// TIA Portal V17 export
// export: Created 2025-03-05T08:01:46.0565803Z, ExportSetting WithDefaults, DisplayName Totally Integrated Automation Portal, DisplayVersion V17 Update 8, DisplayName TIA Portal Openness, DisplayVersion V17 Update 8, DisplayName TIA Portal Version Control Interface, DisplayVersion V17, DisplayName SINAMICS Startdrive Advanced, DisplayVersion V17 SP2, DisplayName SINAMICS Startdrive G110M, G120, G120C, G120D, G120P, G115D, DisplayVersion V17 SP2, DisplayName SINAMICS Startdrive G130, G150, S120, S150, SINAMICS MV, S210, DisplayVersion V17 SP2, DisplayName STEP 7 Professional, DisplayVersion V17 Update 8, DisplayName SINUMERIK ONE STEP 7 Toolbox, DisplayVersion V17 Update 12, DisplayName SINUMERIK 840D sl STEP 7 Toolbox, DisplayVersion V17 Update 12, DisplayName STEP 7 Safety, DisplayVersion V17 Update 6, DisplayName WinCC Advanced, DisplayVersion V17 Update 8
FUNCTION "FC7240_MACHINE_DEVICE_ENABLE_DISABLE" : Void   // FC7240, LAD
{ S7_Optimized_Access := 'FALSE' }
AUTHOR : ETXETAR
VERSION : 1.0
// stored: AutoNumber false, IsIECCheckEnabled false, SetENOAutomatically false, UDAEnableTagReadback false
BEGIN

REGION Network 1: OPTIONS OFF
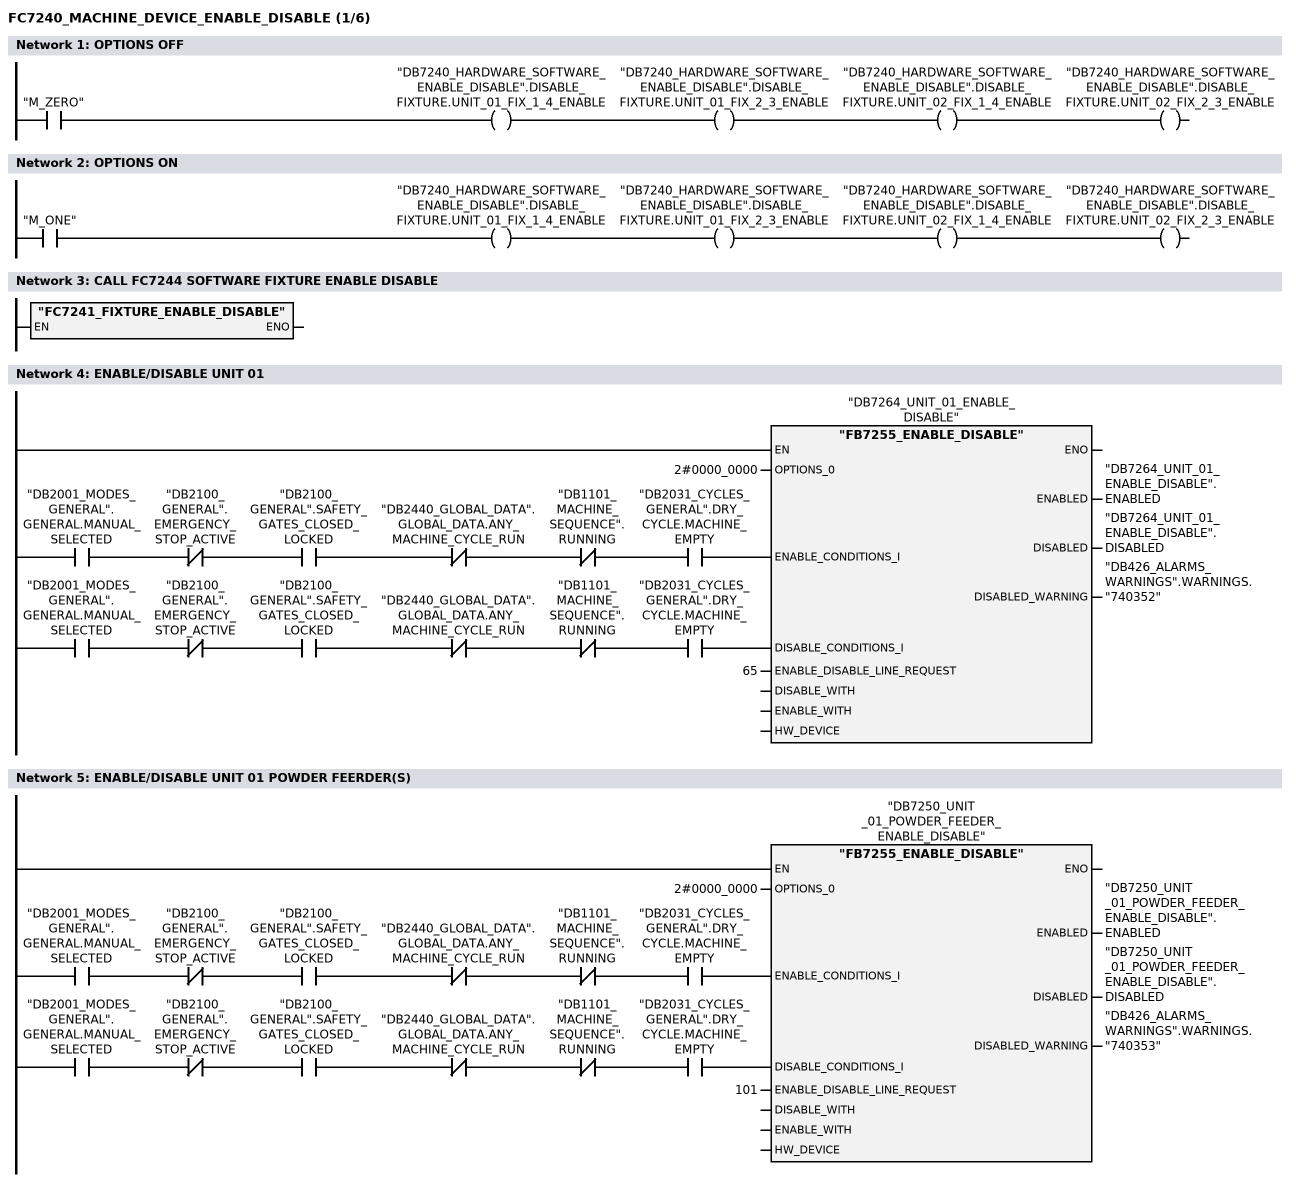
   RUNG wire#powerrail
      Contact( "M_ZERO" )
      Coil( "DB7240_HARDWARE_SOFTWARE_ENABLE_DISABLE".DISABLE_FIXTURE.UNIT_01_FIX_1_4_ENABLE )
      Coil( "DB7240_HARDWARE_SOFTWARE_ENABLE_DISABLE".DISABLE_FIXTURE.UNIT_01_FIX_2_3_ENABLE )
      Coil( "DB7240_HARDWARE_SOFTWARE_ENABLE_DISABLE".DISABLE_FIXTURE.UNIT_02_FIX_1_4_ENABLE )
      Coil( "DB7240_HARDWARE_SOFTWARE_ENABLE_DISABLE".DISABLE_FIXTURE.UNIT_02_FIX_2_3_ENABLE )
   END_RUNG
   // the same network as SCL:
   "DB7240_HARDWARE_SOFTWARE_ENABLE_DISABLE".DISABLE_FIXTURE.UNIT_01_FIX_1_4_ENABLE := "M_ZERO";
   "DB7240_HARDWARE_SOFTWARE_ENABLE_DISABLE".DISABLE_FIXTURE.UNIT_01_FIX_2_3_ENABLE := "M_ZERO";
   "DB7240_HARDWARE_SOFTWARE_ENABLE_DISABLE".DISABLE_FIXTURE.UNIT_02_FIX_1_4_ENABLE := "M_ZERO";
   "DB7240_HARDWARE_SOFTWARE_ENABLE_DISABLE".DISABLE_FIXTURE.UNIT_02_FIX_2_3_ENABLE := "M_ZERO";
END_REGION

REGION Network 2: OPTIONS ON
   RUNG wire#powerrail
      Contact( "M_ONE" )
      Coil( "DB7240_HARDWARE_SOFTWARE_ENABLE_DISABLE".DISABLE_FIXTURE.UNIT_01_FIX_1_4_ENABLE )
      Coil( "DB7240_HARDWARE_SOFTWARE_ENABLE_DISABLE".DISABLE_FIXTURE.UNIT_01_FIX_2_3_ENABLE )
      Coil( "DB7240_HARDWARE_SOFTWARE_ENABLE_DISABLE".DISABLE_FIXTURE.UNIT_02_FIX_1_4_ENABLE )
      Coil( "DB7240_HARDWARE_SOFTWARE_ENABLE_DISABLE".DISABLE_FIXTURE.UNIT_02_FIX_2_3_ENABLE )
   END_RUNG
   // the same network as SCL:
   "DB7240_HARDWARE_SOFTWARE_ENABLE_DISABLE".DISABLE_FIXTURE.UNIT_01_FIX_1_4_ENABLE := "M_ONE";
   "DB7240_HARDWARE_SOFTWARE_ENABLE_DISABLE".DISABLE_FIXTURE.UNIT_01_FIX_2_3_ENABLE := "M_ONE";
   "DB7240_HARDWARE_SOFTWARE_ENABLE_DISABLE".DISABLE_FIXTURE.UNIT_02_FIX_1_4_ENABLE := "M_ONE";
   "DB7240_HARDWARE_SOFTWARE_ENABLE_DISABLE".DISABLE_FIXTURE.UNIT_02_FIX_2_3_ENABLE := "M_ONE";
END_REGION

REGION Network 3: CALL FC7244 SOFTWARE FIXTURE ENABLE DISABLE
   RUNG wire#powerrail
      "FC7241_FIXTURE_ENABLE_DISABLE"()
   END_RUNG
   // the same network as SCL:
   "FC7241_FIXTURE_ENABLE_DISABLE"();
END_REGION

REGION Network 4: ENABLE/DISABLE UNIT 01
   RUNG wire#powerrail
      "DB7264_UNIT_01_ENABLE_DISABLE"(ENABLE_CONDITIONS_I := wire#w1, DISABLE_CONDITIONS_I := wire#w2, OPTIONS_0 := 2#0000_0000, ENABLE_DISABLE_LINE_REQUEST := 65, DISABLE_WITH :=, ENABLE_WITH :=, HW_DEVICE :=, ENABLED => "DB7264_UNIT_01_ENABLE_DISABLE".ENABLED, DISABLED => "DB7264_UNIT_01_ENABLE_DISABLE".DISABLED, DISABLED_WARNING => "DB426_ALARMS_WARNINGS".WARNINGS."740352")
   END_RUNG
   RUNG wire#powerrail
      Contact( "DB2001_MODES_GENERAL".GENERAL.MANUAL_SELECTED )
      I_Contact( "DB2100_GENERAL".EMERGENCY_STOP_ACTIVE )
      Contact( "DB2100_GENERAL".SAFETY_GATES_CLOSED_LOCKED )
      I_Contact( "DB2440_GLOBAL_DATA".GLOBAL_DATA.ANY_MACHINE_CYCLE_RUN )
      I_Contact( "DB1101_MACHINE_SEQUENCE".RUNNING )
      Contact( "DB2031_CYCLES_GENERAL".DRY_CYCLE.MACHINE_EMPTY )
   END_RUNG wire#w1
   RUNG wire#powerrail
      Contact( "DB2001_MODES_GENERAL".GENERAL.MANUAL_SELECTED )
      I_Contact( "DB2100_GENERAL".EMERGENCY_STOP_ACTIVE )
      Contact( "DB2100_GENERAL".SAFETY_GATES_CLOSED_LOCKED )
      I_Contact( "DB2440_GLOBAL_DATA".GLOBAL_DATA.ANY_MACHINE_CYCLE_RUN )
      I_Contact( "DB1101_MACHINE_SEQUENCE".RUNNING )
      Contact( "DB2031_CYCLES_GENERAL".DRY_CYCLE.MACHINE_EMPTY )
   END_RUNG wire#w2
   // the same network as SCL:
   "DB7264_UNIT_01_ENABLE_DISABLE"(OPTIONS_0 := 2#0000_0000,   // "FB7255_ENABLE_DISABLE"
                           ENABLE_CONDITIONS_I := "DB2001_MODES_GENERAL".GENERAL.MANUAL_SELECTED AND NOT "DB2100_GENERAL".EMERGENCY_STOP_ACTIVE AND "DB2100_GENERAL".SAFETY_GATES_CLOSED_LOCKED AND NOT "DB2440_GLOBAL_DATA".GLOBAL_DATA.ANY_MACHINE_CYCLE_RUN AND NOT "DB1101_MACHINE_SEQUENCE".RUNNING AND "DB2031_CYCLES_GENERAL".DRY_CYCLE.MACHINE_EMPTY,
                           DISABLE_CONDITIONS_I := "DB2001_MODES_GENERAL".GENERAL.MANUAL_SELECTED AND NOT "DB2100_GENERAL".EMERGENCY_STOP_ACTIVE AND "DB2100_GENERAL".SAFETY_GATES_CLOSED_LOCKED AND NOT "DB2440_GLOBAL_DATA".GLOBAL_DATA.ANY_MACHINE_CYCLE_RUN AND NOT "DB1101_MACHINE_SEQUENCE".RUNNING AND "DB2031_CYCLES_GENERAL".DRY_CYCLE.MACHINE_EMPTY,
                           ENABLE_DISABLE_LINE_REQUEST := 65,
                           ENABLED => "DB7264_UNIT_01_ENABLE_DISABLE".ENABLED,
                           DISABLED => "DB7264_UNIT_01_ENABLE_DISABLE".DISABLED,
                           DISABLED_WARNING => "DB426_ALARMS_WARNINGS".WARNINGS."740352");
END_REGION

REGION Network 5: ENABLE/DISABLE UNIT 01 POWDER FEERDER(S)
   RUNG wire#powerrail
      "DB7250_UNIT _01_POWDER_FEEDER_ENABLE_DISABLE"(ENABLE_CONDITIONS_I := wire#w1, DISABLE_CONDITIONS_I := wire#w2, OPTIONS_0 := 2#0000_0000, ENABLE_DISABLE_LINE_REQUEST := 101, DISABLE_WITH :=, ENABLE_WITH :=, HW_DEVICE :=, ENABLED => "DB7250_UNIT _01_POWDER_FEEDER_ENABLE_DISABLE".ENABLED, DISABLED => "DB7250_UNIT _01_POWDER_FEEDER_ENABLE_DISABLE".DISABLED, DISABLED_WARNING => "DB426_ALARMS_WARNINGS".WARNINGS."740353")
   END_RUNG
   RUNG wire#powerrail
      Contact( "DB2001_MODES_GENERAL".GENERAL.MANUAL_SELECTED )
      I_Contact( "DB2100_GENERAL".EMERGENCY_STOP_ACTIVE )
      Contact( "DB2100_GENERAL".SAFETY_GATES_CLOSED_LOCKED )
      I_Contact( "DB2440_GLOBAL_DATA".GLOBAL_DATA.ANY_MACHINE_CYCLE_RUN )
      I_Contact( "DB1101_MACHINE_SEQUENCE".RUNNING )
      Contact( "DB2031_CYCLES_GENERAL".DRY_CYCLE.MACHINE_EMPTY )
   END_RUNG wire#w1
   RUNG wire#powerrail
      Contact( "DB2001_MODES_GENERAL".GENERAL.MANUAL_SELECTED )
      I_Contact( "DB2100_GENERAL".EMERGENCY_STOP_ACTIVE )
      Contact( "DB2100_GENERAL".SAFETY_GATES_CLOSED_LOCKED )
      I_Contact( "DB2440_GLOBAL_DATA".GLOBAL_DATA.ANY_MACHINE_CYCLE_RUN )
      I_Contact( "DB1101_MACHINE_SEQUENCE".RUNNING )
      Contact( "DB2031_CYCLES_GENERAL".DRY_CYCLE.MACHINE_EMPTY )
   END_RUNG wire#w2
   // the same network as SCL:
   "DB7250_UNIT _01_POWDER_FEEDER_ENABLE_DISABLE"(OPTIONS_0 := 2#0000_0000,   // "FB7255_ENABLE_DISABLE"
                           ENABLE_CONDITIONS_I := "DB2001_MODES_GENERAL".GENERAL.MANUAL_SELECTED AND NOT "DB2100_GENERAL".EMERGENCY_STOP_ACTIVE AND "DB2100_GENERAL".SAFETY_GATES_CLOSED_LOCKED AND NOT "DB2440_GLOBAL_DATA".GLOBAL_DATA.ANY_MACHINE_CYCLE_RUN AND NOT "DB1101_MACHINE_SEQUENCE".RUNNING AND "DB2031_CYCLES_GENERAL".DRY_CYCLE.MACHINE_EMPTY,
                           DISABLE_CONDITIONS_I := "DB2001_MODES_GENERAL".GENERAL.MANUAL_SELECTED AND NOT "DB2100_GENERAL".EMERGENCY_STOP_ACTIVE AND "DB2100_GENERAL".SAFETY_GATES_CLOSED_LOCKED AND NOT "DB2440_GLOBAL_DATA".GLOBAL_DATA.ANY_MACHINE_CYCLE_RUN AND NOT "DB1101_MACHINE_SEQUENCE".RUNNING AND "DB2031_CYCLES_GENERAL".DRY_CYCLE.MACHINE_EMPTY,
                           ENABLE_DISABLE_LINE_REQUEST := 101,
                           ENABLED => "DB7250_UNIT _01_POWDER_FEEDER_ENABLE_DISABLE".ENABLED,
                           DISABLED => "DB7250_UNIT _01_POWDER_FEEDER_ENABLE_DISABLE".DISABLED,
                           DISABLED_WARNING => "DB426_ALARMS_WARNINGS".WARNINGS."740353");
END_REGION

REGION Network 6: ENABLE/DISABLE UNIT 01 PYROMETER
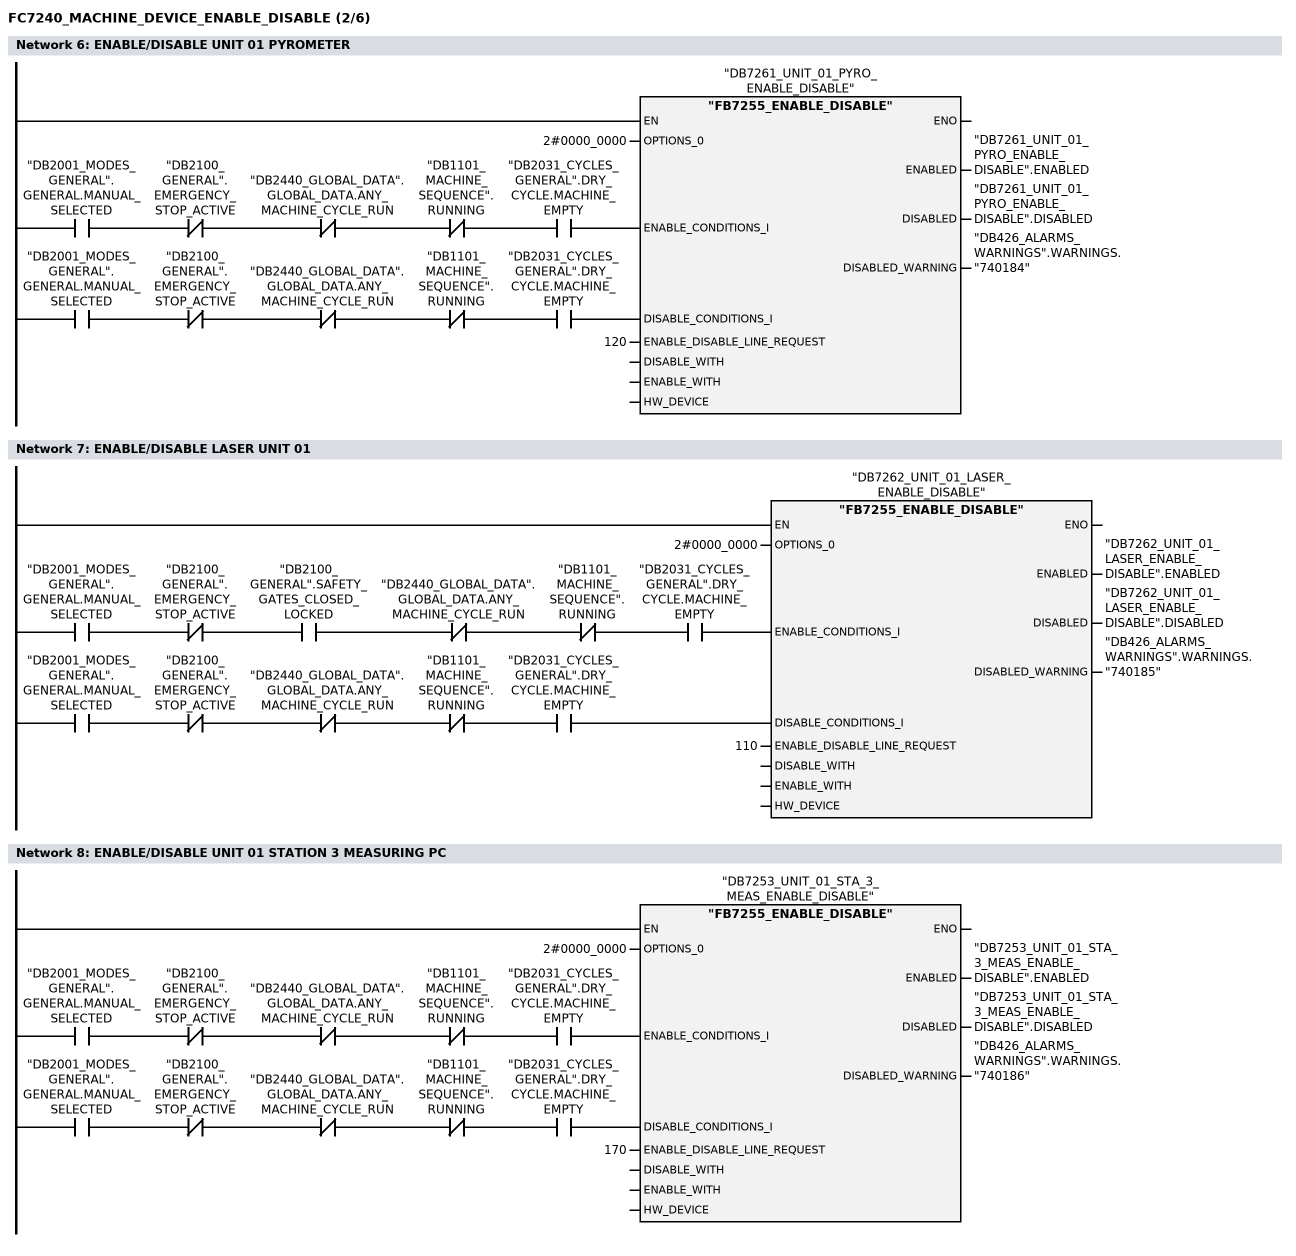
   RUNG wire#powerrail
      "DB7261_UNIT_01_PYRO_ENABLE_DISABLE"(ENABLE_CONDITIONS_I := wire#w1, DISABLE_CONDITIONS_I := wire#w2, OPTIONS_0 := 2#0000_0000, ENABLE_DISABLE_LINE_REQUEST := 120, DISABLE_WITH :=, ENABLE_WITH :=, HW_DEVICE :=, ENABLED => "DB7261_UNIT_01_PYRO_ENABLE_DISABLE".ENABLED, DISABLED => "DB7261_UNIT_01_PYRO_ENABLE_DISABLE".DISABLED, DISABLED_WARNING => "DB426_ALARMS_WARNINGS".WARNINGS."740184")
   END_RUNG
   RUNG wire#powerrail
      Contact( "DB2001_MODES_GENERAL".GENERAL.MANUAL_SELECTED )
      I_Contact( "DB2100_GENERAL".EMERGENCY_STOP_ACTIVE )
      I_Contact( "DB2440_GLOBAL_DATA".GLOBAL_DATA.ANY_MACHINE_CYCLE_RUN )
      I_Contact( "DB1101_MACHINE_SEQUENCE".RUNNING )
      Contact( "DB2031_CYCLES_GENERAL".DRY_CYCLE.MACHINE_EMPTY )
   END_RUNG wire#w1
   RUNG wire#powerrail
      Contact( "DB2001_MODES_GENERAL".GENERAL.MANUAL_SELECTED )
      I_Contact( "DB2100_GENERAL".EMERGENCY_STOP_ACTIVE )
      I_Contact( "DB2440_GLOBAL_DATA".GLOBAL_DATA.ANY_MACHINE_CYCLE_RUN )
      I_Contact( "DB1101_MACHINE_SEQUENCE".RUNNING )
      Contact( "DB2031_CYCLES_GENERAL".DRY_CYCLE.MACHINE_EMPTY )
   END_RUNG wire#w2
   // the same network as SCL:
   "DB7261_UNIT_01_PYRO_ENABLE_DISABLE"(OPTIONS_0 := 2#0000_0000,   // "FB7255_ENABLE_DISABLE"
                           ENABLE_CONDITIONS_I := "DB2001_MODES_GENERAL".GENERAL.MANUAL_SELECTED AND NOT "DB2100_GENERAL".EMERGENCY_STOP_ACTIVE AND NOT "DB2440_GLOBAL_DATA".GLOBAL_DATA.ANY_MACHINE_CYCLE_RUN AND NOT "DB1101_MACHINE_SEQUENCE".RUNNING AND "DB2031_CYCLES_GENERAL".DRY_CYCLE.MACHINE_EMPTY,
                           DISABLE_CONDITIONS_I := "DB2001_MODES_GENERAL".GENERAL.MANUAL_SELECTED AND NOT "DB2100_GENERAL".EMERGENCY_STOP_ACTIVE AND NOT "DB2440_GLOBAL_DATA".GLOBAL_DATA.ANY_MACHINE_CYCLE_RUN AND NOT "DB1101_MACHINE_SEQUENCE".RUNNING AND "DB2031_CYCLES_GENERAL".DRY_CYCLE.MACHINE_EMPTY,
                           ENABLE_DISABLE_LINE_REQUEST := 120,
                           ENABLED => "DB7261_UNIT_01_PYRO_ENABLE_DISABLE".ENABLED,
                           DISABLED => "DB7261_UNIT_01_PYRO_ENABLE_DISABLE".DISABLED,
                           DISABLED_WARNING => "DB426_ALARMS_WARNINGS".WARNINGS."740184");
END_REGION

REGION Network 7: ENABLE/DISABLE LASER UNIT 01
   RUNG wire#powerrail
      "DB7262_UNIT_01_LASER_ENABLE_DISABLE"(ENABLE_CONDITIONS_I := wire#w1, DISABLE_CONDITIONS_I := wire#w2, OPTIONS_0 := 2#0000_0000, ENABLE_DISABLE_LINE_REQUEST := 110, DISABLE_WITH :=, ENABLE_WITH :=, HW_DEVICE :=, ENABLED => "DB7262_UNIT_01_LASER_ENABLE_DISABLE".ENABLED, DISABLED => "DB7262_UNIT_01_LASER_ENABLE_DISABLE".DISABLED, DISABLED_WARNING => "DB426_ALARMS_WARNINGS".WARNINGS."740185")
   END_RUNG
   RUNG wire#powerrail
      Contact( "DB2001_MODES_GENERAL".GENERAL.MANUAL_SELECTED )
      I_Contact( "DB2100_GENERAL".EMERGENCY_STOP_ACTIVE )
      Contact( "DB2100_GENERAL".SAFETY_GATES_CLOSED_LOCKED )
      I_Contact( "DB2440_GLOBAL_DATA".GLOBAL_DATA.ANY_MACHINE_CYCLE_RUN )
      I_Contact( "DB1101_MACHINE_SEQUENCE".RUNNING )
      Contact( "DB2031_CYCLES_GENERAL".DRY_CYCLE.MACHINE_EMPTY )
   END_RUNG wire#w1
   RUNG wire#powerrail
      Contact( "DB2001_MODES_GENERAL".GENERAL.MANUAL_SELECTED )
      I_Contact( "DB2100_GENERAL".EMERGENCY_STOP_ACTIVE )
      I_Contact( "DB2440_GLOBAL_DATA".GLOBAL_DATA.ANY_MACHINE_CYCLE_RUN )
      I_Contact( "DB1101_MACHINE_SEQUENCE".RUNNING )
      Contact( "DB2031_CYCLES_GENERAL".DRY_CYCLE.MACHINE_EMPTY )
   END_RUNG wire#w2
   // the same network as SCL:
   "DB7262_UNIT_01_LASER_ENABLE_DISABLE"(OPTIONS_0 := 2#0000_0000,   // "FB7255_ENABLE_DISABLE"
                           ENABLE_CONDITIONS_I := "DB2001_MODES_GENERAL".GENERAL.MANUAL_SELECTED AND NOT "DB2100_GENERAL".EMERGENCY_STOP_ACTIVE AND "DB2100_GENERAL".SAFETY_GATES_CLOSED_LOCKED AND NOT "DB2440_GLOBAL_DATA".GLOBAL_DATA.ANY_MACHINE_CYCLE_RUN AND NOT "DB1101_MACHINE_SEQUENCE".RUNNING AND "DB2031_CYCLES_GENERAL".DRY_CYCLE.MACHINE_EMPTY,
                           DISABLE_CONDITIONS_I := "DB2001_MODES_GENERAL".GENERAL.MANUAL_SELECTED AND NOT "DB2100_GENERAL".EMERGENCY_STOP_ACTIVE AND NOT "DB2440_GLOBAL_DATA".GLOBAL_DATA.ANY_MACHINE_CYCLE_RUN AND NOT "DB1101_MACHINE_SEQUENCE".RUNNING AND "DB2031_CYCLES_GENERAL".DRY_CYCLE.MACHINE_EMPTY,
                           ENABLE_DISABLE_LINE_REQUEST := 110,
                           ENABLED => "DB7262_UNIT_01_LASER_ENABLE_DISABLE".ENABLED,
                           DISABLED => "DB7262_UNIT_01_LASER_ENABLE_DISABLE".DISABLED,
                           DISABLED_WARNING => "DB426_ALARMS_WARNINGS".WARNINGS."740185");
END_REGION

REGION Network 8: ENABLE/DISABLE UNIT 01 STATION 3 MEASURING PC
   RUNG wire#powerrail
      "DB7253_UNIT_01_STA_3_MEAS_ENABLE_DISABLE"(ENABLE_CONDITIONS_I := wire#w1, DISABLE_CONDITIONS_I := wire#w2, OPTIONS_0 := 2#0000_0000, ENABLE_DISABLE_LINE_REQUEST := 170, DISABLE_WITH :=, ENABLE_WITH :=, HW_DEVICE :=, ENABLED => "DB7253_UNIT_01_STA_3_MEAS_ENABLE_DISABLE".ENABLED, DISABLED => "DB7253_UNIT_01_STA_3_MEAS_ENABLE_DISABLE".DISABLED, DISABLED_WARNING => "DB426_ALARMS_WARNINGS".WARNINGS."740186")
   END_RUNG
   RUNG wire#powerrail
      Contact( "DB2001_MODES_GENERAL".GENERAL.MANUAL_SELECTED )
      I_Contact( "DB2100_GENERAL".EMERGENCY_STOP_ACTIVE )
      I_Contact( "DB2440_GLOBAL_DATA".GLOBAL_DATA.ANY_MACHINE_CYCLE_RUN )
      I_Contact( "DB1101_MACHINE_SEQUENCE".RUNNING )
      Contact( "DB2031_CYCLES_GENERAL".DRY_CYCLE.MACHINE_EMPTY )
   END_RUNG wire#w1
   RUNG wire#powerrail
      Contact( "DB2001_MODES_GENERAL".GENERAL.MANUAL_SELECTED )
      I_Contact( "DB2100_GENERAL".EMERGENCY_STOP_ACTIVE )
      I_Contact( "DB2440_GLOBAL_DATA".GLOBAL_DATA.ANY_MACHINE_CYCLE_RUN )
      I_Contact( "DB1101_MACHINE_SEQUENCE".RUNNING )
      Contact( "DB2031_CYCLES_GENERAL".DRY_CYCLE.MACHINE_EMPTY )
   END_RUNG wire#w2
   // the same network as SCL:
   "DB7253_UNIT_01_STA_3_MEAS_ENABLE_DISABLE"(OPTIONS_0 := 2#0000_0000,   // "FB7255_ENABLE_DISABLE"
                           ENABLE_CONDITIONS_I := "DB2001_MODES_GENERAL".GENERAL.MANUAL_SELECTED AND NOT "DB2100_GENERAL".EMERGENCY_STOP_ACTIVE AND NOT "DB2440_GLOBAL_DATA".GLOBAL_DATA.ANY_MACHINE_CYCLE_RUN AND NOT "DB1101_MACHINE_SEQUENCE".RUNNING AND "DB2031_CYCLES_GENERAL".DRY_CYCLE.MACHINE_EMPTY,
                           DISABLE_CONDITIONS_I := "DB2001_MODES_GENERAL".GENERAL.MANUAL_SELECTED AND NOT "DB2100_GENERAL".EMERGENCY_STOP_ACTIVE AND NOT "DB2440_GLOBAL_DATA".GLOBAL_DATA.ANY_MACHINE_CYCLE_RUN AND NOT "DB1101_MACHINE_SEQUENCE".RUNNING AND "DB2031_CYCLES_GENERAL".DRY_CYCLE.MACHINE_EMPTY,
                           ENABLE_DISABLE_LINE_REQUEST := 170,
                           ENABLED => "DB7253_UNIT_01_STA_3_MEAS_ENABLE_DISABLE".ENABLED,
                           DISABLED => "DB7253_UNIT_01_STA_3_MEAS_ENABLE_DISABLE".DISABLED,
                           DISABLED_WARNING => "DB426_ALARMS_WARNINGS".WARNINGS."740186");
END_REGION

REGION Network 9: ENABLE/DISABLE UNIT 01 STATION 3 COAXIAL PC
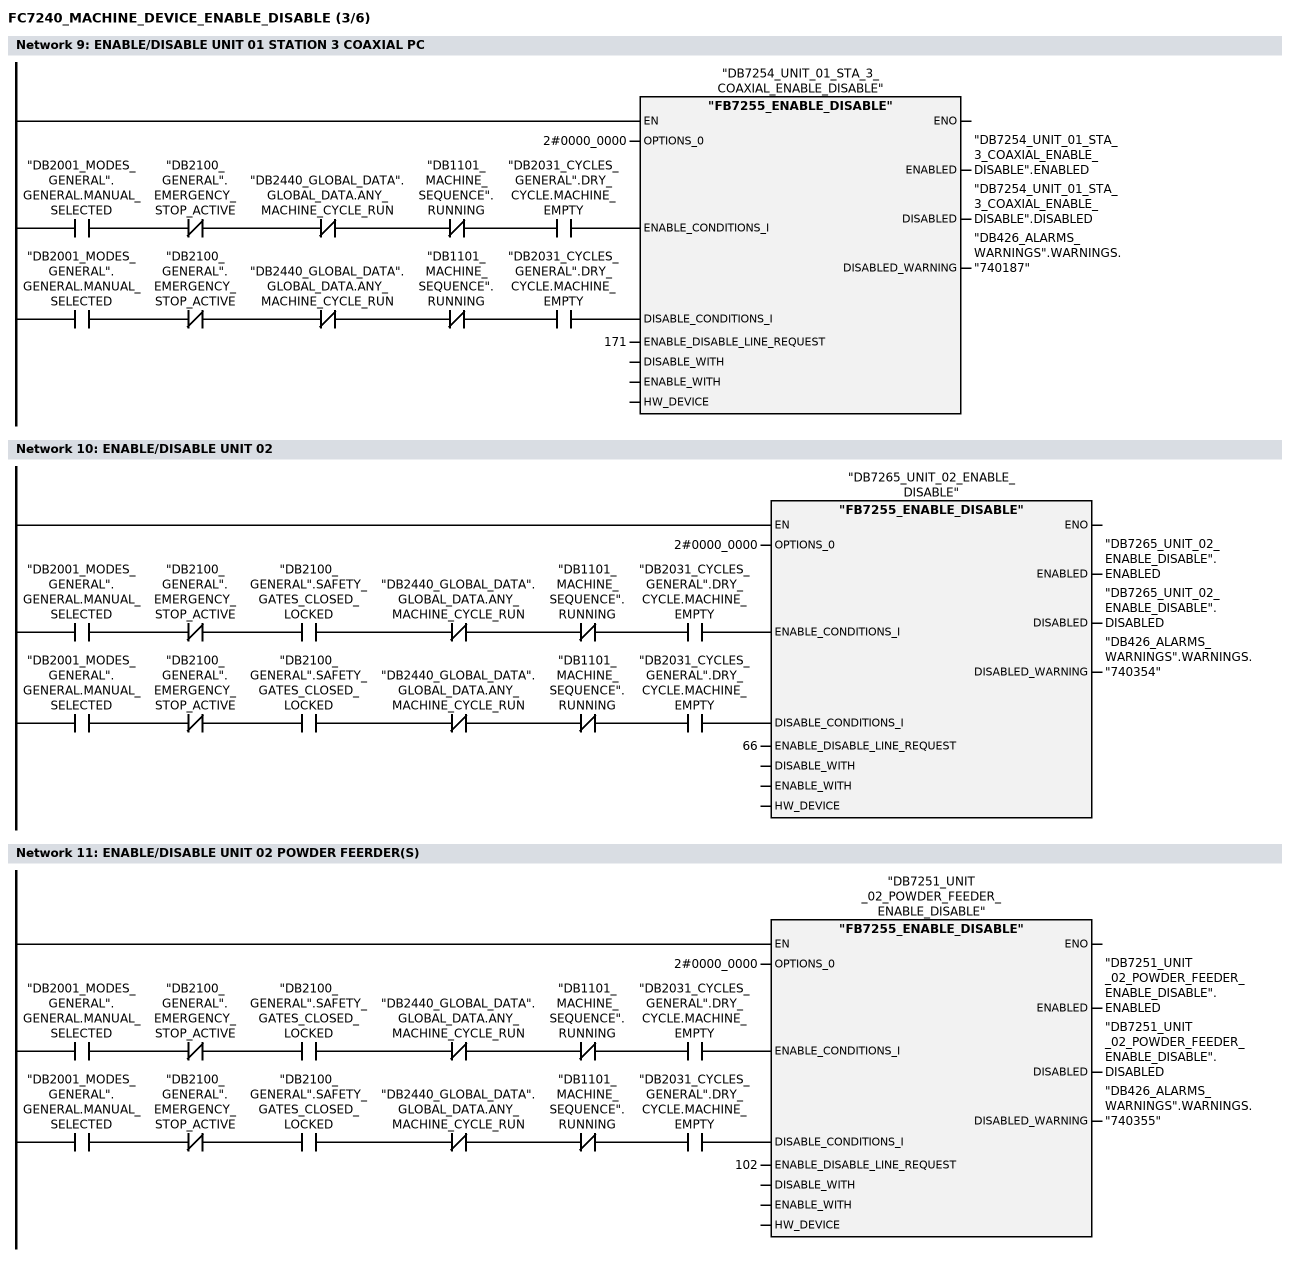
   RUNG wire#powerrail
      "DB7254_UNIT_01_STA_3_COAXIAL_ENABLE_DISABLE"(ENABLE_CONDITIONS_I := wire#w1, DISABLE_CONDITIONS_I := wire#w2, OPTIONS_0 := 2#0000_0000, ENABLE_DISABLE_LINE_REQUEST := 171, DISABLE_WITH :=, ENABLE_WITH :=, HW_DEVICE :=, ENABLED => "DB7254_UNIT_01_STA_3_COAXIAL_ENABLE_DISABLE".ENABLED, DISABLED => "DB7254_UNIT_01_STA_3_COAXIAL_ENABLE_DISABLE".DISABLED, DISABLED_WARNING => "DB426_ALARMS_WARNINGS".WARNINGS."740187")
   END_RUNG
   RUNG wire#powerrail
      Contact( "DB2001_MODES_GENERAL".GENERAL.MANUAL_SELECTED )
      I_Contact( "DB2100_GENERAL".EMERGENCY_STOP_ACTIVE )
      I_Contact( "DB2440_GLOBAL_DATA".GLOBAL_DATA.ANY_MACHINE_CYCLE_RUN )
      I_Contact( "DB1101_MACHINE_SEQUENCE".RUNNING )
      Contact( "DB2031_CYCLES_GENERAL".DRY_CYCLE.MACHINE_EMPTY )
   END_RUNG wire#w1
   RUNG wire#powerrail
      Contact( "DB2001_MODES_GENERAL".GENERAL.MANUAL_SELECTED )
      I_Contact( "DB2100_GENERAL".EMERGENCY_STOP_ACTIVE )
      I_Contact( "DB2440_GLOBAL_DATA".GLOBAL_DATA.ANY_MACHINE_CYCLE_RUN )
      I_Contact( "DB1101_MACHINE_SEQUENCE".RUNNING )
      Contact( "DB2031_CYCLES_GENERAL".DRY_CYCLE.MACHINE_EMPTY )
   END_RUNG wire#w2
   // the same network as SCL:
   "DB7254_UNIT_01_STA_3_COAXIAL_ENABLE_DISABLE"(OPTIONS_0 := 2#0000_0000,   // "FB7255_ENABLE_DISABLE"
                           ENABLE_CONDITIONS_I := "DB2001_MODES_GENERAL".GENERAL.MANUAL_SELECTED AND NOT "DB2100_GENERAL".EMERGENCY_STOP_ACTIVE AND NOT "DB2440_GLOBAL_DATA".GLOBAL_DATA.ANY_MACHINE_CYCLE_RUN AND NOT "DB1101_MACHINE_SEQUENCE".RUNNING AND "DB2031_CYCLES_GENERAL".DRY_CYCLE.MACHINE_EMPTY,
                           DISABLE_CONDITIONS_I := "DB2001_MODES_GENERAL".GENERAL.MANUAL_SELECTED AND NOT "DB2100_GENERAL".EMERGENCY_STOP_ACTIVE AND NOT "DB2440_GLOBAL_DATA".GLOBAL_DATA.ANY_MACHINE_CYCLE_RUN AND NOT "DB1101_MACHINE_SEQUENCE".RUNNING AND "DB2031_CYCLES_GENERAL".DRY_CYCLE.MACHINE_EMPTY,
                           ENABLE_DISABLE_LINE_REQUEST := 171,
                           ENABLED => "DB7254_UNIT_01_STA_3_COAXIAL_ENABLE_DISABLE".ENABLED,
                           DISABLED => "DB7254_UNIT_01_STA_3_COAXIAL_ENABLE_DISABLE".DISABLED,
                           DISABLED_WARNING => "DB426_ALARMS_WARNINGS".WARNINGS."740187");
END_REGION

REGION Network 10: ENABLE/DISABLE UNIT 02
   RUNG wire#powerrail
      "DB7265_UNIT_02_ENABLE_DISABLE"(ENABLE_CONDITIONS_I := wire#w1, DISABLE_CONDITIONS_I := wire#w2, OPTIONS_0 := 2#0000_0000, ENABLE_DISABLE_LINE_REQUEST := 66, DISABLE_WITH :=, ENABLE_WITH :=, HW_DEVICE :=, ENABLED => "DB7265_UNIT_02_ENABLE_DISABLE".ENABLED, DISABLED => "DB7265_UNIT_02_ENABLE_DISABLE".DISABLED, DISABLED_WARNING => "DB426_ALARMS_WARNINGS".WARNINGS."740354")
   END_RUNG
   RUNG wire#powerrail
      Contact( "DB2001_MODES_GENERAL".GENERAL.MANUAL_SELECTED )
      I_Contact( "DB2100_GENERAL".EMERGENCY_STOP_ACTIVE )
      Contact( "DB2100_GENERAL".SAFETY_GATES_CLOSED_LOCKED )
      I_Contact( "DB2440_GLOBAL_DATA".GLOBAL_DATA.ANY_MACHINE_CYCLE_RUN )
      I_Contact( "DB1101_MACHINE_SEQUENCE".RUNNING )
      Contact( "DB2031_CYCLES_GENERAL".DRY_CYCLE.MACHINE_EMPTY )
   END_RUNG wire#w1
   RUNG wire#powerrail
      Contact( "DB2001_MODES_GENERAL".GENERAL.MANUAL_SELECTED )
      I_Contact( "DB2100_GENERAL".EMERGENCY_STOP_ACTIVE )
      Contact( "DB2100_GENERAL".SAFETY_GATES_CLOSED_LOCKED )
      I_Contact( "DB2440_GLOBAL_DATA".GLOBAL_DATA.ANY_MACHINE_CYCLE_RUN )
      I_Contact( "DB1101_MACHINE_SEQUENCE".RUNNING )
      Contact( "DB2031_CYCLES_GENERAL".DRY_CYCLE.MACHINE_EMPTY )
   END_RUNG wire#w2
   // the same network as SCL:
   "DB7265_UNIT_02_ENABLE_DISABLE"(OPTIONS_0 := 2#0000_0000,   // "FB7255_ENABLE_DISABLE"
                           ENABLE_CONDITIONS_I := "DB2001_MODES_GENERAL".GENERAL.MANUAL_SELECTED AND NOT "DB2100_GENERAL".EMERGENCY_STOP_ACTIVE AND "DB2100_GENERAL".SAFETY_GATES_CLOSED_LOCKED AND NOT "DB2440_GLOBAL_DATA".GLOBAL_DATA.ANY_MACHINE_CYCLE_RUN AND NOT "DB1101_MACHINE_SEQUENCE".RUNNING AND "DB2031_CYCLES_GENERAL".DRY_CYCLE.MACHINE_EMPTY,
                           DISABLE_CONDITIONS_I := "DB2001_MODES_GENERAL".GENERAL.MANUAL_SELECTED AND NOT "DB2100_GENERAL".EMERGENCY_STOP_ACTIVE AND "DB2100_GENERAL".SAFETY_GATES_CLOSED_LOCKED AND NOT "DB2440_GLOBAL_DATA".GLOBAL_DATA.ANY_MACHINE_CYCLE_RUN AND NOT "DB1101_MACHINE_SEQUENCE".RUNNING AND "DB2031_CYCLES_GENERAL".DRY_CYCLE.MACHINE_EMPTY,
                           ENABLE_DISABLE_LINE_REQUEST := 66,
                           ENABLED => "DB7265_UNIT_02_ENABLE_DISABLE".ENABLED,
                           DISABLED => "DB7265_UNIT_02_ENABLE_DISABLE".DISABLED,
                           DISABLED_WARNING => "DB426_ALARMS_WARNINGS".WARNINGS."740354");
END_REGION

REGION Network 11: ENABLE/DISABLE UNIT 02 POWDER FEERDER(S)
   RUNG wire#powerrail
      "DB7251_UNIT _02_POWDER_FEEDER_ENABLE_DISABLE"(ENABLE_CONDITIONS_I := wire#w1, DISABLE_CONDITIONS_I := wire#w2, OPTIONS_0 := 2#0000_0000, ENABLE_DISABLE_LINE_REQUEST := 102, DISABLE_WITH :=, ENABLE_WITH :=, HW_DEVICE :=, ENABLED => "DB7251_UNIT _02_POWDER_FEEDER_ENABLE_DISABLE".ENABLED, DISABLED => "DB7251_UNIT _02_POWDER_FEEDER_ENABLE_DISABLE".DISABLED, DISABLED_WARNING => "DB426_ALARMS_WARNINGS".WARNINGS."740355")
   END_RUNG
   RUNG wire#powerrail
      Contact( "DB2001_MODES_GENERAL".GENERAL.MANUAL_SELECTED )
      I_Contact( "DB2100_GENERAL".EMERGENCY_STOP_ACTIVE )
      Contact( "DB2100_GENERAL".SAFETY_GATES_CLOSED_LOCKED )
      I_Contact( "DB2440_GLOBAL_DATA".GLOBAL_DATA.ANY_MACHINE_CYCLE_RUN )
      I_Contact( "DB1101_MACHINE_SEQUENCE".RUNNING )
      Contact( "DB2031_CYCLES_GENERAL".DRY_CYCLE.MACHINE_EMPTY )
   END_RUNG wire#w1
   RUNG wire#powerrail
      Contact( "DB2001_MODES_GENERAL".GENERAL.MANUAL_SELECTED )
      I_Contact( "DB2100_GENERAL".EMERGENCY_STOP_ACTIVE )
      Contact( "DB2100_GENERAL".SAFETY_GATES_CLOSED_LOCKED )
      I_Contact( "DB2440_GLOBAL_DATA".GLOBAL_DATA.ANY_MACHINE_CYCLE_RUN )
      I_Contact( "DB1101_MACHINE_SEQUENCE".RUNNING )
      Contact( "DB2031_CYCLES_GENERAL".DRY_CYCLE.MACHINE_EMPTY )
   END_RUNG wire#w2
   // the same network as SCL:
   "DB7251_UNIT _02_POWDER_FEEDER_ENABLE_DISABLE"(OPTIONS_0 := 2#0000_0000,   // "FB7255_ENABLE_DISABLE"
                           ENABLE_CONDITIONS_I := "DB2001_MODES_GENERAL".GENERAL.MANUAL_SELECTED AND NOT "DB2100_GENERAL".EMERGENCY_STOP_ACTIVE AND "DB2100_GENERAL".SAFETY_GATES_CLOSED_LOCKED AND NOT "DB2440_GLOBAL_DATA".GLOBAL_DATA.ANY_MACHINE_CYCLE_RUN AND NOT "DB1101_MACHINE_SEQUENCE".RUNNING AND "DB2031_CYCLES_GENERAL".DRY_CYCLE.MACHINE_EMPTY,
                           DISABLE_CONDITIONS_I := "DB2001_MODES_GENERAL".GENERAL.MANUAL_SELECTED AND NOT "DB2100_GENERAL".EMERGENCY_STOP_ACTIVE AND "DB2100_GENERAL".SAFETY_GATES_CLOSED_LOCKED AND NOT "DB2440_GLOBAL_DATA".GLOBAL_DATA.ANY_MACHINE_CYCLE_RUN AND NOT "DB1101_MACHINE_SEQUENCE".RUNNING AND "DB2031_CYCLES_GENERAL".DRY_CYCLE.MACHINE_EMPTY,
                           ENABLE_DISABLE_LINE_REQUEST := 102,
                           ENABLED => "DB7251_UNIT _02_POWDER_FEEDER_ENABLE_DISABLE".ENABLED,
                           DISABLED => "DB7251_UNIT _02_POWDER_FEEDER_ENABLE_DISABLE".DISABLED,
                           DISABLED_WARNING => "DB426_ALARMS_WARNINGS".WARNINGS."740355");
END_REGION

REGION Network 12: ENABLE/DISABLE UNIT 02 STATION 2 MEASURING PC
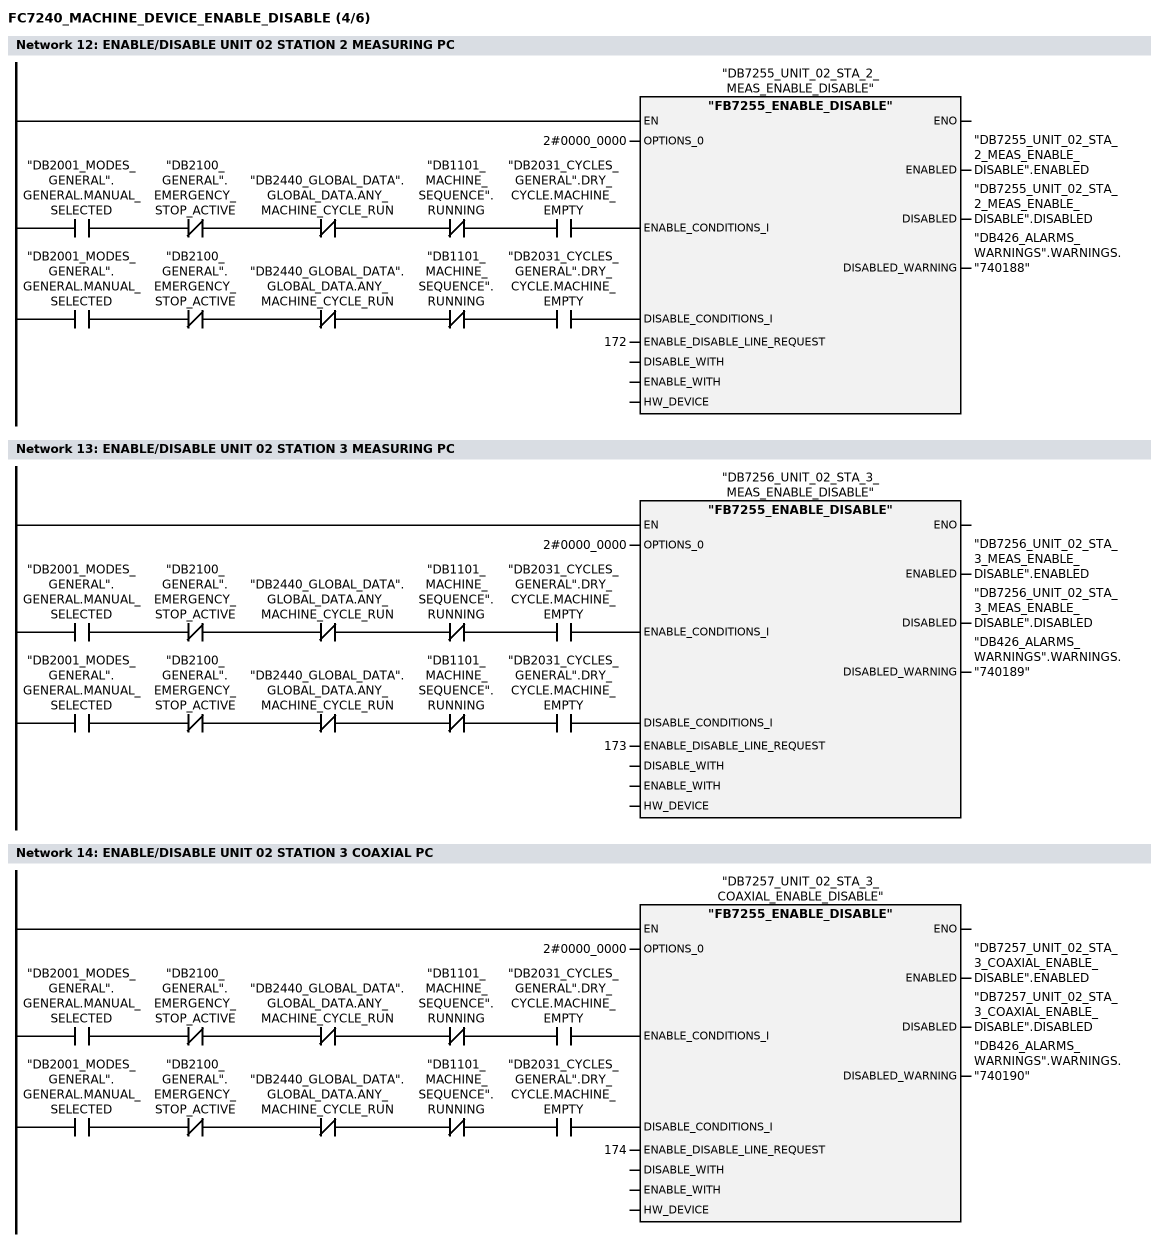
   RUNG wire#powerrail
      "DB7255_UNIT_02_STA_2_MEAS_ENABLE_DISABLE"(ENABLE_CONDITIONS_I := wire#w1, DISABLE_CONDITIONS_I := wire#w2, OPTIONS_0 := 2#0000_0000, ENABLE_DISABLE_LINE_REQUEST := 172, DISABLE_WITH :=, ENABLE_WITH :=, HW_DEVICE :=, ENABLED => "DB7255_UNIT_02_STA_2_MEAS_ENABLE_DISABLE".ENABLED, DISABLED => "DB7255_UNIT_02_STA_2_MEAS_ENABLE_DISABLE".DISABLED, DISABLED_WARNING => "DB426_ALARMS_WARNINGS".WARNINGS."740188")
   END_RUNG
   RUNG wire#powerrail
      Contact( "DB2001_MODES_GENERAL".GENERAL.MANUAL_SELECTED )
      I_Contact( "DB2100_GENERAL".EMERGENCY_STOP_ACTIVE )
      I_Contact( "DB2440_GLOBAL_DATA".GLOBAL_DATA.ANY_MACHINE_CYCLE_RUN )
      I_Contact( "DB1101_MACHINE_SEQUENCE".RUNNING )
      Contact( "DB2031_CYCLES_GENERAL".DRY_CYCLE.MACHINE_EMPTY )
   END_RUNG wire#w1
   RUNG wire#powerrail
      Contact( "DB2001_MODES_GENERAL".GENERAL.MANUAL_SELECTED )
      I_Contact( "DB2100_GENERAL".EMERGENCY_STOP_ACTIVE )
      I_Contact( "DB2440_GLOBAL_DATA".GLOBAL_DATA.ANY_MACHINE_CYCLE_RUN )
      I_Contact( "DB1101_MACHINE_SEQUENCE".RUNNING )
      Contact( "DB2031_CYCLES_GENERAL".DRY_CYCLE.MACHINE_EMPTY )
   END_RUNG wire#w2
   // the same network as SCL:
   "DB7255_UNIT_02_STA_2_MEAS_ENABLE_DISABLE"(OPTIONS_0 := 2#0000_0000,   // "FB7255_ENABLE_DISABLE"
                           ENABLE_CONDITIONS_I := "DB2001_MODES_GENERAL".GENERAL.MANUAL_SELECTED AND NOT "DB2100_GENERAL".EMERGENCY_STOP_ACTIVE AND NOT "DB2440_GLOBAL_DATA".GLOBAL_DATA.ANY_MACHINE_CYCLE_RUN AND NOT "DB1101_MACHINE_SEQUENCE".RUNNING AND "DB2031_CYCLES_GENERAL".DRY_CYCLE.MACHINE_EMPTY,
                           DISABLE_CONDITIONS_I := "DB2001_MODES_GENERAL".GENERAL.MANUAL_SELECTED AND NOT "DB2100_GENERAL".EMERGENCY_STOP_ACTIVE AND NOT "DB2440_GLOBAL_DATA".GLOBAL_DATA.ANY_MACHINE_CYCLE_RUN AND NOT "DB1101_MACHINE_SEQUENCE".RUNNING AND "DB2031_CYCLES_GENERAL".DRY_CYCLE.MACHINE_EMPTY,
                           ENABLE_DISABLE_LINE_REQUEST := 172,
                           ENABLED => "DB7255_UNIT_02_STA_2_MEAS_ENABLE_DISABLE".ENABLED,
                           DISABLED => "DB7255_UNIT_02_STA_2_MEAS_ENABLE_DISABLE".DISABLED,
                           DISABLED_WARNING => "DB426_ALARMS_WARNINGS".WARNINGS."740188");
END_REGION

REGION Network 13: ENABLE/DISABLE UNIT 02 STATION 3 MEASURING PC
   RUNG wire#powerrail
      "DB7256_UNIT_02_STA_3_MEAS_ENABLE_DISABLE"(ENABLE_CONDITIONS_I := wire#w1, DISABLE_CONDITIONS_I := wire#w2, OPTIONS_0 := 2#0000_0000, ENABLE_DISABLE_LINE_REQUEST := 173, DISABLE_WITH :=, ENABLE_WITH :=, HW_DEVICE :=, ENABLED => "DB7256_UNIT_02_STA_3_MEAS_ENABLE_DISABLE".ENABLED, DISABLED => "DB7256_UNIT_02_STA_3_MEAS_ENABLE_DISABLE".DISABLED, DISABLED_WARNING => "DB426_ALARMS_WARNINGS".WARNINGS."740189")
   END_RUNG
   RUNG wire#powerrail
      Contact( "DB2001_MODES_GENERAL".GENERAL.MANUAL_SELECTED )
      I_Contact( "DB2100_GENERAL".EMERGENCY_STOP_ACTIVE )
      I_Contact( "DB2440_GLOBAL_DATA".GLOBAL_DATA.ANY_MACHINE_CYCLE_RUN )
      I_Contact( "DB1101_MACHINE_SEQUENCE".RUNNING )
      Contact( "DB2031_CYCLES_GENERAL".DRY_CYCLE.MACHINE_EMPTY )
   END_RUNG wire#w1
   RUNG wire#powerrail
      Contact( "DB2001_MODES_GENERAL".GENERAL.MANUAL_SELECTED )
      I_Contact( "DB2100_GENERAL".EMERGENCY_STOP_ACTIVE )
      I_Contact( "DB2440_GLOBAL_DATA".GLOBAL_DATA.ANY_MACHINE_CYCLE_RUN )
      I_Contact( "DB1101_MACHINE_SEQUENCE".RUNNING )
      Contact( "DB2031_CYCLES_GENERAL".DRY_CYCLE.MACHINE_EMPTY )
   END_RUNG wire#w2
   // the same network as SCL:
   "DB7256_UNIT_02_STA_3_MEAS_ENABLE_DISABLE"(OPTIONS_0 := 2#0000_0000,   // "FB7255_ENABLE_DISABLE"
                           ENABLE_CONDITIONS_I := "DB2001_MODES_GENERAL".GENERAL.MANUAL_SELECTED AND NOT "DB2100_GENERAL".EMERGENCY_STOP_ACTIVE AND NOT "DB2440_GLOBAL_DATA".GLOBAL_DATA.ANY_MACHINE_CYCLE_RUN AND NOT "DB1101_MACHINE_SEQUENCE".RUNNING AND "DB2031_CYCLES_GENERAL".DRY_CYCLE.MACHINE_EMPTY,
                           DISABLE_CONDITIONS_I := "DB2001_MODES_GENERAL".GENERAL.MANUAL_SELECTED AND NOT "DB2100_GENERAL".EMERGENCY_STOP_ACTIVE AND NOT "DB2440_GLOBAL_DATA".GLOBAL_DATA.ANY_MACHINE_CYCLE_RUN AND NOT "DB1101_MACHINE_SEQUENCE".RUNNING AND "DB2031_CYCLES_GENERAL".DRY_CYCLE.MACHINE_EMPTY,
                           ENABLE_DISABLE_LINE_REQUEST := 173,
                           ENABLED => "DB7256_UNIT_02_STA_3_MEAS_ENABLE_DISABLE".ENABLED,
                           DISABLED => "DB7256_UNIT_02_STA_3_MEAS_ENABLE_DISABLE".DISABLED,
                           DISABLED_WARNING => "DB426_ALARMS_WARNINGS".WARNINGS."740189");
END_REGION

REGION Network 14: ENABLE/DISABLE UNIT 02 STATION 3 COAXIAL PC
   RUNG wire#powerrail
      "DB7257_UNIT_02_STA_3_COAXIAL_ENABLE_DISABLE"(ENABLE_CONDITIONS_I := wire#w1, DISABLE_CONDITIONS_I := wire#w2, OPTIONS_0 := 2#0000_0000, ENABLE_DISABLE_LINE_REQUEST := 174, DISABLE_WITH :=, ENABLE_WITH :=, HW_DEVICE :=, ENABLED => "DB7257_UNIT_02_STA_3_COAXIAL_ENABLE_DISABLE".ENABLED, DISABLED => "DB7257_UNIT_02_STA_3_COAXIAL_ENABLE_DISABLE".DISABLED, DISABLED_WARNING => "DB426_ALARMS_WARNINGS".WARNINGS."740190")
   END_RUNG
   RUNG wire#powerrail
      Contact( "DB2001_MODES_GENERAL".GENERAL.MANUAL_SELECTED )
      I_Contact( "DB2100_GENERAL".EMERGENCY_STOP_ACTIVE )
      I_Contact( "DB2440_GLOBAL_DATA".GLOBAL_DATA.ANY_MACHINE_CYCLE_RUN )
      I_Contact( "DB1101_MACHINE_SEQUENCE".RUNNING )
      Contact( "DB2031_CYCLES_GENERAL".DRY_CYCLE.MACHINE_EMPTY )
   END_RUNG wire#w1
   RUNG wire#powerrail
      Contact( "DB2001_MODES_GENERAL".GENERAL.MANUAL_SELECTED )
      I_Contact( "DB2100_GENERAL".EMERGENCY_STOP_ACTIVE )
      I_Contact( "DB2440_GLOBAL_DATA".GLOBAL_DATA.ANY_MACHINE_CYCLE_RUN )
      I_Contact( "DB1101_MACHINE_SEQUENCE".RUNNING )
      Contact( "DB2031_CYCLES_GENERAL".DRY_CYCLE.MACHINE_EMPTY )
   END_RUNG wire#w2
   // the same network as SCL:
   "DB7257_UNIT_02_STA_3_COAXIAL_ENABLE_DISABLE"(OPTIONS_0 := 2#0000_0000,   // "FB7255_ENABLE_DISABLE"
                           ENABLE_CONDITIONS_I := "DB2001_MODES_GENERAL".GENERAL.MANUAL_SELECTED AND NOT "DB2100_GENERAL".EMERGENCY_STOP_ACTIVE AND NOT "DB2440_GLOBAL_DATA".GLOBAL_DATA.ANY_MACHINE_CYCLE_RUN AND NOT "DB1101_MACHINE_SEQUENCE".RUNNING AND "DB2031_CYCLES_GENERAL".DRY_CYCLE.MACHINE_EMPTY,
                           DISABLE_CONDITIONS_I := "DB2001_MODES_GENERAL".GENERAL.MANUAL_SELECTED AND NOT "DB2100_GENERAL".EMERGENCY_STOP_ACTIVE AND NOT "DB2440_GLOBAL_DATA".GLOBAL_DATA.ANY_MACHINE_CYCLE_RUN AND NOT "DB1101_MACHINE_SEQUENCE".RUNNING AND "DB2031_CYCLES_GENERAL".DRY_CYCLE.MACHINE_EMPTY,
                           ENABLE_DISABLE_LINE_REQUEST := 174,
                           ENABLED => "DB7257_UNIT_02_STA_3_COAXIAL_ENABLE_DISABLE".ENABLED,
                           DISABLED => "DB7257_UNIT_02_STA_3_COAXIAL_ENABLE_DISABLE".DISABLED,
                           DISABLED_WARNING => "DB426_ALARMS_WARNINGS".WARNINGS."740190");
END_REGION

REGION Network 15: ENABLE/DISABLE LASER UNIT 02
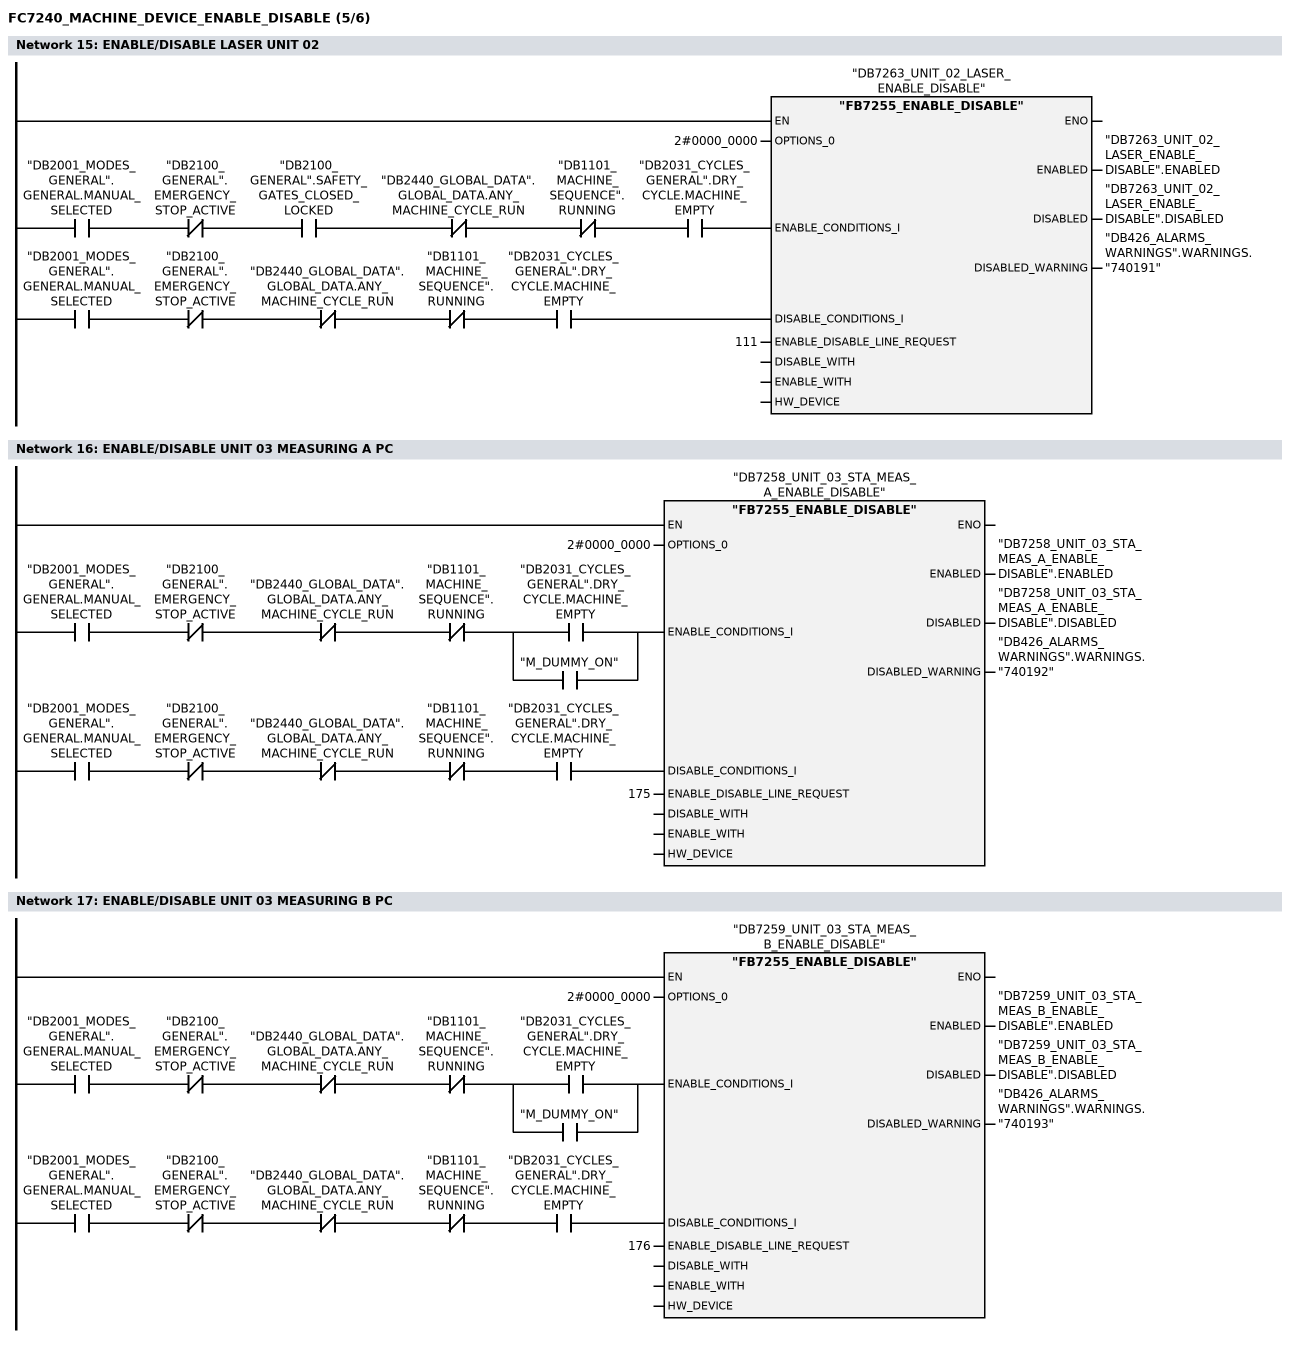
   RUNG wire#powerrail
      "DB7263_UNIT_02_LASER_ENABLE_DISABLE"(ENABLE_CONDITIONS_I := wire#w1, DISABLE_CONDITIONS_I := wire#w2, OPTIONS_0 := 2#0000_0000, ENABLE_DISABLE_LINE_REQUEST := 111, DISABLE_WITH :=, ENABLE_WITH :=, HW_DEVICE :=, ENABLED => "DB7263_UNIT_02_LASER_ENABLE_DISABLE".ENABLED, DISABLED => "DB7263_UNIT_02_LASER_ENABLE_DISABLE".DISABLED, DISABLED_WARNING => "DB426_ALARMS_WARNINGS".WARNINGS."740191")
   END_RUNG
   RUNG wire#powerrail
      Contact( "DB2001_MODES_GENERAL".GENERAL.MANUAL_SELECTED )
      I_Contact( "DB2100_GENERAL".EMERGENCY_STOP_ACTIVE )
      Contact( "DB2100_GENERAL".SAFETY_GATES_CLOSED_LOCKED )
      I_Contact( "DB2440_GLOBAL_DATA".GLOBAL_DATA.ANY_MACHINE_CYCLE_RUN )
      I_Contact( "DB1101_MACHINE_SEQUENCE".RUNNING )
      Contact( "DB2031_CYCLES_GENERAL".DRY_CYCLE.MACHINE_EMPTY )
   END_RUNG wire#w1
   RUNG wire#powerrail
      Contact( "DB2001_MODES_GENERAL".GENERAL.MANUAL_SELECTED )
      I_Contact( "DB2100_GENERAL".EMERGENCY_STOP_ACTIVE )
      I_Contact( "DB2440_GLOBAL_DATA".GLOBAL_DATA.ANY_MACHINE_CYCLE_RUN )
      I_Contact( "DB1101_MACHINE_SEQUENCE".RUNNING )
      Contact( "DB2031_CYCLES_GENERAL".DRY_CYCLE.MACHINE_EMPTY )
   END_RUNG wire#w2
   // the same network as SCL:
   "DB7263_UNIT_02_LASER_ENABLE_DISABLE"(OPTIONS_0 := 2#0000_0000,   // "FB7255_ENABLE_DISABLE"
                           ENABLE_CONDITIONS_I := "DB2001_MODES_GENERAL".GENERAL.MANUAL_SELECTED AND NOT "DB2100_GENERAL".EMERGENCY_STOP_ACTIVE AND "DB2100_GENERAL".SAFETY_GATES_CLOSED_LOCKED AND NOT "DB2440_GLOBAL_DATA".GLOBAL_DATA.ANY_MACHINE_CYCLE_RUN AND NOT "DB1101_MACHINE_SEQUENCE".RUNNING AND "DB2031_CYCLES_GENERAL".DRY_CYCLE.MACHINE_EMPTY,
                           DISABLE_CONDITIONS_I := "DB2001_MODES_GENERAL".GENERAL.MANUAL_SELECTED AND NOT "DB2100_GENERAL".EMERGENCY_STOP_ACTIVE AND NOT "DB2440_GLOBAL_DATA".GLOBAL_DATA.ANY_MACHINE_CYCLE_RUN AND NOT "DB1101_MACHINE_SEQUENCE".RUNNING AND "DB2031_CYCLES_GENERAL".DRY_CYCLE.MACHINE_EMPTY,
                           ENABLE_DISABLE_LINE_REQUEST := 111,
                           ENABLED => "DB7263_UNIT_02_LASER_ENABLE_DISABLE".ENABLED,
                           DISABLED => "DB7263_UNIT_02_LASER_ENABLE_DISABLE".DISABLED,
                           DISABLED_WARNING => "DB426_ALARMS_WARNINGS".WARNINGS."740191");
END_REGION

REGION Network 16: ENABLE/DISABLE UNIT 03 MEASURING A PC
   RUNG wire#powerrail
      "DB7258_UNIT_03_STA_MEAS_A_ENABLE_DISABLE"(ENABLE_CONDITIONS_I := wire#w2, DISABLE_CONDITIONS_I := wire#w3, OPTIONS_0 := 2#0000_0000, ENABLE_DISABLE_LINE_REQUEST := 175, DISABLE_WITH :=, ENABLE_WITH :=, HW_DEVICE :=, ENABLED => "DB7258_UNIT_03_STA_MEAS_A_ENABLE_DISABLE".ENABLED, DISABLED => "DB7258_UNIT_03_STA_MEAS_A_ENABLE_DISABLE".DISABLED, DISABLED_WARNING => "DB426_ALARMS_WARNINGS".WARNINGS."740192")
   END_RUNG
   RUNG wire#powerrail
      Contact( "DB2001_MODES_GENERAL".GENERAL.MANUAL_SELECTED )
      I_Contact( "DB2100_GENERAL".EMERGENCY_STOP_ACTIVE )
      I_Contact( "DB2440_GLOBAL_DATA".GLOBAL_DATA.ANY_MACHINE_CYCLE_RUN )
      I_Contact( "DB1101_MACHINE_SEQUENCE".RUNNING )
      wire#w1
      Contact( "DB2031_CYCLES_GENERAL".DRY_CYCLE.MACHINE_EMPTY )
   END_RUNG wire#w2
   RUNG wire#w1
      Contact( "M_DUMMY_ON" )
   END_RUNG wire#w2
   RUNG wire#powerrail
      Contact( "DB2001_MODES_GENERAL".GENERAL.MANUAL_SELECTED )
      I_Contact( "DB2100_GENERAL".EMERGENCY_STOP_ACTIVE )
      I_Contact( "DB2440_GLOBAL_DATA".GLOBAL_DATA.ANY_MACHINE_CYCLE_RUN )
      I_Contact( "DB1101_MACHINE_SEQUENCE".RUNNING )
      Contact( "DB2031_CYCLES_GENERAL".DRY_CYCLE.MACHINE_EMPTY )
   END_RUNG wire#w3
   // the same network as SCL:
   "DB7258_UNIT_03_STA_MEAS_A_ENABLE_DISABLE"(OPTIONS_0 := 2#0000_0000,   // "FB7255_ENABLE_DISABLE"
                           ENABLE_CONDITIONS_I := "DB2001_MODES_GENERAL".GENERAL.MANUAL_SELECTED AND NOT "DB2100_GENERAL".EMERGENCY_STOP_ACTIVE AND NOT "DB2440_GLOBAL_DATA".GLOBAL_DATA.ANY_MACHINE_CYCLE_RUN AND NOT "DB1101_MACHINE_SEQUENCE".RUNNING AND ("DB2031_CYCLES_GENERAL".DRY_CYCLE.MACHINE_EMPTY OR "M_DUMMY_ON"),
                           DISABLE_CONDITIONS_I := "DB2001_MODES_GENERAL".GENERAL.MANUAL_SELECTED AND NOT "DB2100_GENERAL".EMERGENCY_STOP_ACTIVE AND NOT "DB2440_GLOBAL_DATA".GLOBAL_DATA.ANY_MACHINE_CYCLE_RUN AND NOT "DB1101_MACHINE_SEQUENCE".RUNNING AND "DB2031_CYCLES_GENERAL".DRY_CYCLE.MACHINE_EMPTY,
                           ENABLE_DISABLE_LINE_REQUEST := 175,
                           ENABLED => "DB7258_UNIT_03_STA_MEAS_A_ENABLE_DISABLE".ENABLED,
                           DISABLED => "DB7258_UNIT_03_STA_MEAS_A_ENABLE_DISABLE".DISABLED,
                           DISABLED_WARNING => "DB426_ALARMS_WARNINGS".WARNINGS."740192");
END_REGION

REGION Network 17: ENABLE/DISABLE UNIT 03 MEASURING B PC
   RUNG wire#powerrail
      "DB7259_UNIT_03_STA_MEAS_B_ENABLE_DISABLE"(ENABLE_CONDITIONS_I := wire#w2, DISABLE_CONDITIONS_I := wire#w3, OPTIONS_0 := 2#0000_0000, ENABLE_DISABLE_LINE_REQUEST := 176, DISABLE_WITH :=, ENABLE_WITH :=, HW_DEVICE :=, ENABLED => "DB7259_UNIT_03_STA_MEAS_B_ENABLE_DISABLE".ENABLED, DISABLED => "DB7259_UNIT_03_STA_MEAS_B_ENABLE_DISABLE".DISABLED, DISABLED_WARNING => "DB426_ALARMS_WARNINGS".WARNINGS."740193")
   END_RUNG
   RUNG wire#powerrail
      Contact( "DB2001_MODES_GENERAL".GENERAL.MANUAL_SELECTED )
      I_Contact( "DB2100_GENERAL".EMERGENCY_STOP_ACTIVE )
      I_Contact( "DB2440_GLOBAL_DATA".GLOBAL_DATA.ANY_MACHINE_CYCLE_RUN )
      I_Contact( "DB1101_MACHINE_SEQUENCE".RUNNING )
      wire#w1
      Contact( "DB2031_CYCLES_GENERAL".DRY_CYCLE.MACHINE_EMPTY )
   END_RUNG wire#w2
   RUNG wire#w1
      Contact( "M_DUMMY_ON" )
   END_RUNG wire#w2
   RUNG wire#powerrail
      Contact( "DB2001_MODES_GENERAL".GENERAL.MANUAL_SELECTED )
      I_Contact( "DB2100_GENERAL".EMERGENCY_STOP_ACTIVE )
      I_Contact( "DB2440_GLOBAL_DATA".GLOBAL_DATA.ANY_MACHINE_CYCLE_RUN )
      I_Contact( "DB1101_MACHINE_SEQUENCE".RUNNING )
      Contact( "DB2031_CYCLES_GENERAL".DRY_CYCLE.MACHINE_EMPTY )
   END_RUNG wire#w3
   // the same network as SCL:
   "DB7259_UNIT_03_STA_MEAS_B_ENABLE_DISABLE"(OPTIONS_0 := 2#0000_0000,   // "FB7255_ENABLE_DISABLE"
                           ENABLE_CONDITIONS_I := "DB2001_MODES_GENERAL".GENERAL.MANUAL_SELECTED AND NOT "DB2100_GENERAL".EMERGENCY_STOP_ACTIVE AND NOT "DB2440_GLOBAL_DATA".GLOBAL_DATA.ANY_MACHINE_CYCLE_RUN AND NOT "DB1101_MACHINE_SEQUENCE".RUNNING AND ("DB2031_CYCLES_GENERAL".DRY_CYCLE.MACHINE_EMPTY OR "M_DUMMY_ON"),
                           DISABLE_CONDITIONS_I := "DB2001_MODES_GENERAL".GENERAL.MANUAL_SELECTED AND NOT "DB2100_GENERAL".EMERGENCY_STOP_ACTIVE AND NOT "DB2440_GLOBAL_DATA".GLOBAL_DATA.ANY_MACHINE_CYCLE_RUN AND NOT "DB1101_MACHINE_SEQUENCE".RUNNING AND "DB2031_CYCLES_GENERAL".DRY_CYCLE.MACHINE_EMPTY,
                           ENABLE_DISABLE_LINE_REQUEST := 176,
                           ENABLED => "DB7259_UNIT_03_STA_MEAS_B_ENABLE_DISABLE".ENABLED,
                           DISABLED => "DB7259_UNIT_03_STA_MEAS_B_ENABLE_DISABLE".DISABLED,
                           DISABLED_WARNING => "DB426_ALARMS_WARNINGS".WARNINGS."740193");
END_REGION

REGION Network 18: ENABLE/DISABLE HOLA PC
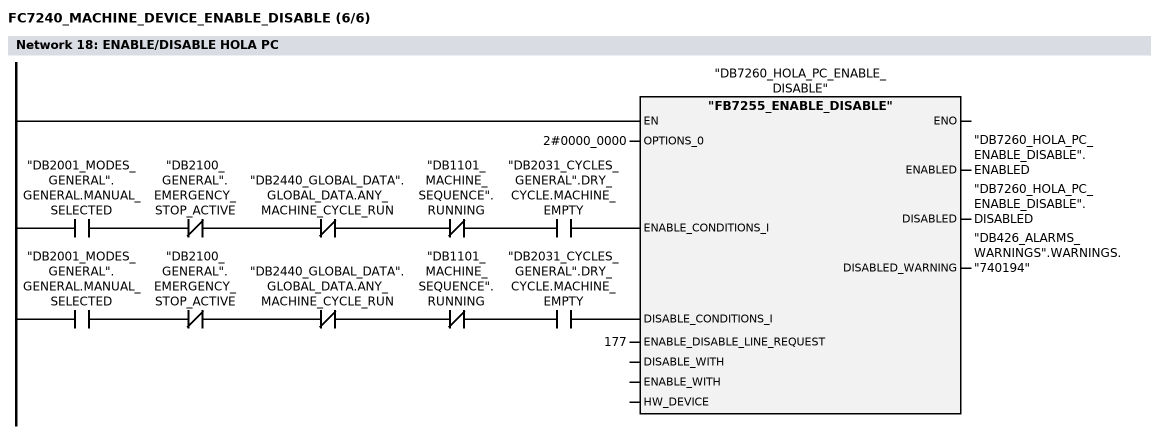
   RUNG wire#powerrail
      "DB7260_HOLA_PC_ENABLE_DISABLE"(ENABLE_CONDITIONS_I := wire#w1, DISABLE_CONDITIONS_I := wire#w2, OPTIONS_0 := 2#0000_0000, ENABLE_DISABLE_LINE_REQUEST := 177, DISABLE_WITH :=, ENABLE_WITH :=, HW_DEVICE :=, ENABLED => "DB7260_HOLA_PC_ENABLE_DISABLE".ENABLED, DISABLED => "DB7260_HOLA_PC_ENABLE_DISABLE".DISABLED, DISABLED_WARNING => "DB426_ALARMS_WARNINGS".WARNINGS."740194")
   END_RUNG
   RUNG wire#powerrail
      Contact( "DB2001_MODES_GENERAL".GENERAL.MANUAL_SELECTED )
      I_Contact( "DB2100_GENERAL".EMERGENCY_STOP_ACTIVE )
      I_Contact( "DB2440_GLOBAL_DATA".GLOBAL_DATA.ANY_MACHINE_CYCLE_RUN )
      I_Contact( "DB1101_MACHINE_SEQUENCE".RUNNING )
      Contact( "DB2031_CYCLES_GENERAL".DRY_CYCLE.MACHINE_EMPTY )
   END_RUNG wire#w1
   RUNG wire#powerrail
      Contact( "DB2001_MODES_GENERAL".GENERAL.MANUAL_SELECTED )
      I_Contact( "DB2100_GENERAL".EMERGENCY_STOP_ACTIVE )
      I_Contact( "DB2440_GLOBAL_DATA".GLOBAL_DATA.ANY_MACHINE_CYCLE_RUN )
      I_Contact( "DB1101_MACHINE_SEQUENCE".RUNNING )
      Contact( "DB2031_CYCLES_GENERAL".DRY_CYCLE.MACHINE_EMPTY )
   END_RUNG wire#w2
   // the same network as SCL:
   "DB7260_HOLA_PC_ENABLE_DISABLE"(OPTIONS_0 := 2#0000_0000,   // "FB7255_ENABLE_DISABLE"
                           ENABLE_CONDITIONS_I := "DB2001_MODES_GENERAL".GENERAL.MANUAL_SELECTED AND NOT "DB2100_GENERAL".EMERGENCY_STOP_ACTIVE AND NOT "DB2440_GLOBAL_DATA".GLOBAL_DATA.ANY_MACHINE_CYCLE_RUN AND NOT "DB1101_MACHINE_SEQUENCE".RUNNING AND "DB2031_CYCLES_GENERAL".DRY_CYCLE.MACHINE_EMPTY,
                           DISABLE_CONDITIONS_I := "DB2001_MODES_GENERAL".GENERAL.MANUAL_SELECTED AND NOT "DB2100_GENERAL".EMERGENCY_STOP_ACTIVE AND NOT "DB2440_GLOBAL_DATA".GLOBAL_DATA.ANY_MACHINE_CYCLE_RUN AND NOT "DB1101_MACHINE_SEQUENCE".RUNNING AND "DB2031_CYCLES_GENERAL".DRY_CYCLE.MACHINE_EMPTY,
                           ENABLE_DISABLE_LINE_REQUEST := 177,
                           ENABLED => "DB7260_HOLA_PC_ENABLE_DISABLE".ENABLED,
                           DISABLED => "DB7260_HOLA_PC_ENABLE_DISABLE".DISABLED,
                           DISABLED_WARNING => "DB426_ALARMS_WARNINGS".WARNINGS."740194");
END_REGION
END_FUNCTION
